Fanuc TP program (LS listing): FOLGE124.LS

/PROG  FOLGE124
/ATTR
OWNER		= AUROM;
COMMENT		= "Mantenimiento";
PROG_SIZE	= 3986;
CREATE		= DATE 03-15-00  TIME 13:37:40;
MODIFIED	= DATE 17-03-12  TIME 11:50:48;
FILE_NAME	= ;
VERSION		= 0;
LINE_COUNT	= 22;
MEMORY_SIZE	= 6070;
PROTECT		= READ_WRITE;
TCD:  STACK_SIZE	= 500,
      TASK_PRIORITY	= 50,
      TIME_SLICE	= 0,
      BUSY_LAMP_OFF	= 0,
      ABORT_REQUEST	= 0,
      PAUSE_REQUEST	= 0;
DEFAULT_GROUP	= 1,1,1,1,*;
CONTROL_CODE	= 00000000 00000000;
/MN
   1:  UTOOL_NUM=1 ;
   2:  UFRAME_NUM=0 ;
   3:  PAYLOAD[1] ;
   4:J P[1] 10% CNT0 ACC100 TB   0.00sec,P-SPS    ;
      1:  IF (DO[12]=ON),CALL MAKRO998 ;
      2:  DO[15]=ON ;
      3:  DO[16]=ON ;
      4:  CALL MAKRO000    ;
      5:  WAIT (DI[9])    ;
       ------ ;
   5:J P[2] 100% CNT0 ACC100 TB   0.00sec,P-SPS    ;
      1:  TC_ONLINE (ON) ;
      2:  DO[23]=OFF ;
      3:  CALL MAKRO050    ;
      4:  !Lib. de Herramientas ;
      5:  DO[80]=ON ;
      6:  DO[78]=OFF ;
      7:  DO[77]=ON ;
      8:  DO[75]=OFF ;
      9:  DO[74]=ON ;
     10:  DO[73]=ON ;
     11:  DO[71]=OFF ;
     12:  DO[70]=OFF ;
     13:  DO[69]=OFF ;
     14:  DO[68]=OFF ;
     15:  DO[67]=OFF ;
     16:  !Lib. de Anticolisiones ;
     17:  DO[41]=ON ;
     18:  DO[42]=ON ;
     19:  DO[43]=ON ;
     20:  DO[44]=ON ;
     21:  DO[45]=ON ;
     22:  DO[46]=ON ;
     23:  !Apagar Posicion Base ;
     24:  DO[15]=OFF ;
     25:  !Garra a Base si no hay pieza ;
     26:  WAIT (M[2])    ;
     27:  F[1]=(ON) ;
     28:  F[3]=(ON) ;
     29:  F[4]=(ON) ;
     30:  F[5]=(ON) ;
     31:  F[6]=(ON) ;
     32:  F[7]=(ON) ;
     33:  IF (!DI[15]),F[17]=(ON) ;
     34:  IF (M[2]),CALL MAKRO342 ;
     35:  CALL MAKRO340    ;
     36:  WAIT (M[31] AND M[35] AND M[37] AND M[39] AND M[41] AND M[43])    ;
     37:  WAIT (DI[23])    ;
     38:  DO[23]=ON ;
     39:  TC_ONLINE (M[2] AND M[30] AND M[31] AND M[35] AND M[37] AND M[39] AND M[41] AND M[43] AND M[95] AND M[96]) ;
       ------ ;
   6:  !Fresado en Mantenimiento ;
   7:J P[3] 100% CNT0 ACC100 TB    .10sec,P-SPS    ;
      1:  TC_ONLINE (ON) ;
      2:  DO[23]=OFF ;
      3:  F[298]=(OFF) ;
      4:  CALL VW_USER(Basic1,EZSP,Nr1 Service,ProgNr=31, , ,S-Punkt=31, ,EIN/AUS=1) ;
      5:  WAIT    .10(sec) ;
      6:  F[79]=((DI[786] AND !DI[788]) OR (!DI[788] AND DI[130])) ;
      7:  F[78]=(DI[788] AND !F[79]) ;
      8:  GO[2]=(R[197]+0) ;
      9:  IF (F[78] OR F[79]),CALL MAKRO085 ;
     10:  IF (F[78] OR F[79]),CALL MAKRO084 ;
     11:  WAIT (M[96])    ;
     12:  WAIT (DI[23])    ;
     13:  DO[23]=ON ;
     14:  TC_ONLINE (M[2] AND M[30] AND M[31] AND M[35] AND M[37] AND M[39] AND M[41] AND M[43] AND M[95] AND M[96]) ;
       ------ ;
   8:  !Pos. de Mantenimiento ;
   9:  !UP112 Mant. G1 ;
  10:  !UP113 Mant. SP1 ;
  11:  !UP201 Cambio Herramienta G1 ;
  12:  !UP202 Cambio Herramienta SP1 ;
  13:  !UP206 TCP Check SP1 ;
  14:J P[4] 100% CNT0 ACC100 TB    .10sec,P-SPS    ;
      1:  TC_ONLINE (ON) ;
      2:  DO[23]=OFF ;
      3:  F[940]=(OFF) ;
      4:  F[941]=(OFF) ;
      5:  F[942]=(OFF) ;
      6:  F[943]=(OFF) ;
      7:  F[944]=(OFF) ;
      8:  WAIT (((DI[20] OR DI[21]) AND (DI[121] OR DI[132])) OR DI[121] OR (DI[132] OR DI[777] OR DI[801]))    ;
      9:  !Mantenimiento G1 ;
     10:  F[940]=(!DI[20] AND !DI[21] AND DI[121] AND !(DI[132] OR DI[777] OR DI[801])) ;
     11:  !Mantenimiento SP1 ;
     12:  F[941]=(!DI[20] AND !DI[21] AND !DI[121] AND (DI[132] OR DI[777] OR DI[801])) ;
     13:  !Cambio de Herramienta G1 ;
     14:  F[942]=(DI[20] AND !DI[21] AND DI[121] AND !DI[132]) ;
     15:  !Cambio de Herramienta SP1 ;
     16:  F[943]=(DI[20] AND !DI[21] AND !DI[121] AND DI[132]) ;
     17:  !TCP Check SP1 ;
     18:  F[944]=(!DI[20] AND DI[21] AND !DI[121] AND DI[132]) ;
     19:  WAIT (F[940] OR F[941] OR F[942] OR F[943] OR F[944])    ;
     20:  WAIT (DI[23])    ;
     21:  DO[23]=ON ;
     22:  TC_ONLINE (M[2] AND M[30] AND M[31] AND M[35] AND M[37] AND M[39] AND M[41] AND M[43] AND M[95] AND M[96]) ;
       ------ ;
  15:  IF (F[940]),CALL UP112 ;
  16:  IF (F[941]),CALL UP113 ;
  17:  IF (F[942]),CALL UP201 ;
  18:  IF (F[943]),CALL UP202 ;
  19:  IF (F[944]),CALL UP206 ;
  20:  UTOOL_NUM=1 ;
  21:  UFRAME_NUM=0 ;
  22:J P[5] 100% CNT0 ACC100 TB   0.00sec,P-SPS    ;
      1:  TC_ONLINE (ON) ;
      2:  DO[15]=ON ;
      3:  DO[14]=ON ;
       ------ ;
/POS
P[1]{
   GP1:
	UF : 0, UT : 1,		CONFIG : 'N U T, 0, 0, 0',
	X =   893.302  mm,	Y =   623.420  mm,	Z =    77.203  mm,
	W =    98.852 deg,	P =    39.834 deg,	R =  -104.177 deg
   GP2:
	UF : 0, UT : 1,
	J1=   100.000  mm
   GP3:
	UF : 0, UT : 1,
	J1=     0.000  mm
   GP4:
	UF : 0, UT : 1,
	J1=     0.000  mm
};
P[2]{
   GP1:
	UF : 0, UT : 1,		CONFIG : 'N U T, 0, 0, 0',
	X =   893.302  mm,	Y =   623.420  mm,	Z =    77.203  mm,
	W =    98.852 deg,	P =    39.834 deg,	R =  -104.177 deg
   GP2:
	UF : 0, UT : 1,
	J1=   100.000  mm
   GP3:
	UF : 0, UT : 1,
	J1=     0.000  mm
   GP4:
	UF : 0, UT : 1,
	J1=     0.000  mm
};
P[3]{
   GP1:
	UF : 0, UT : 1,		CONFIG : 'N U T, 0, 0, 0',
	X =   893.302  mm,	Y =   623.420  mm,	Z =    77.203  mm,
	W =    98.852 deg,	P =    39.834 deg,	R =  -104.177 deg
   GP2:
	UF : 0, UT : 1,
	J1=   100.000  mm
   GP3:
	UF : 0, UT : 1,
	J1=     0.000  mm
   GP4:
	UF : 0, UT : 1,
	J1=     0.000  mm
};
P[4]{
   GP1:
	UF : 0, UT : 1,		CONFIG : 'N U T, 0, 0, 0',
	X =   893.302  mm,	Y =   623.420  mm,	Z =    77.203  mm,
	W =    98.852 deg,	P =    39.834 deg,	R =  -104.177 deg
   GP2:
	UF : 0, UT : 1,
	J1=   100.000  mm
   GP3:
	UF : 0, UT : 1,
	J1=     0.000  mm
   GP4:
	UF : 0, UT : 1,
	J1=     0.000  mm
};
P[5]{
   GP1:
	UF : 0, UT : 1,		CONFIG : 'N U T, 0, 0, 0',
	X =   893.302  mm,	Y =   623.420  mm,	Z =    77.203  mm,
	W =    98.852 deg,	P =    39.834 deg,	R =  -104.177 deg
   GP2:
	UF : 0, UT : 1,
	J1=   100.000  mm
   GP3:
	UF : 0, UT : 1,
	J1=     0.000  mm
   GP4:
	UF : 0, UT : 1,
	J1=     0.000  mm
};
/END
